FUNCTION_BLOCK ConveyorFeed
VAR_INPUT
    Start       : BOOL;
    Stop        : BOOL;
    FaultReset  : BOOL;
END_VAR
VAR_OUTPUT
    Running     : BOOL;
    Faulted     : BOOL;
END_VAR
VAR
    RunningInternal : BOOL;
END_VAR


IF FaultReset THEN
    Faulted := FALSE;
END_IF

IF Start AND NOT Faulted THEN
    RunningInternal := TRUE;
END_IF

IF Stop THEN
    RunningInternal := FALSE;
END_IF

Running := RunningInternal;

END_FUNCTION_BLOCK

(* stored: Version 1.1.0.1, ProductVersion 3.1.4026.18
   POU ConveyorFeed: Id {5177e8e4-938b-477b-ae00-9fe233322905}, SpecialFunc None *)
